// LS Electric XG5000 project: practice1
// PLC LSPLC

PROGRAM NewProgram (task: 스캔 프로그램)

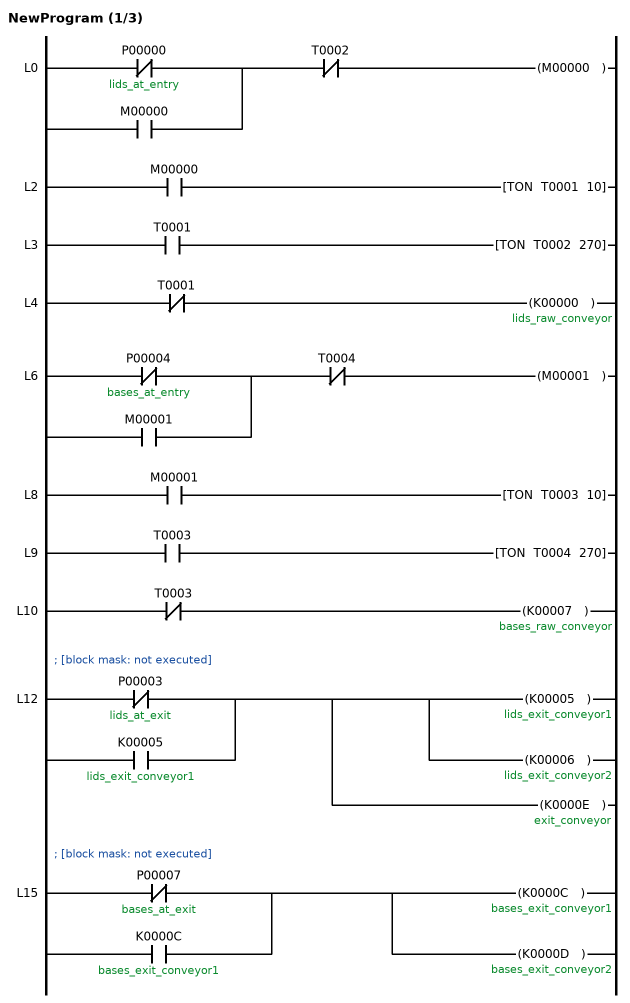
; L0
LOAD NOT  P00000	// lids_at_entry
OR        M00000
AND NOT   T0002
OUT       M00000
; L2
LOAD      M00000
TON       T0001 10
; L3
LOAD      T0001
TON       T0002 270
; L4
LOAD NOT  T0001
OUT       K00000	// lids_raw_conveyor
; L6
LOAD NOT  P00004	// bases_at_entry
OR        M00001
AND NOT   T0004
OUT       M00001
; L8
LOAD      M00001
TON       T0003 10
; L9
LOAD      T0003
TON       T0004 270
; L10
LOAD NOT  T0003
OUT       K00007	// bases_raw_conveyor
; L12 (block mask: not executed)
LOAD NOT  P00003	// lids_at_exit
OR        K00005	// lids_exit_conveyor1
OUT       K00005	// lids_exit_conveyor1
OUT       K00006	// lids_exit_conveyor2
OUT       K0000E	// exit_conveyor
; L15 (block mask: not executed)
LOAD NOT  P00007	// bases_at_exit
OR        K0000C	// bases_exit_conveyor1
OUT       K0000C	// bases_exit_conveyor1
OUT       K0000D	// bases_exit_conveyor2

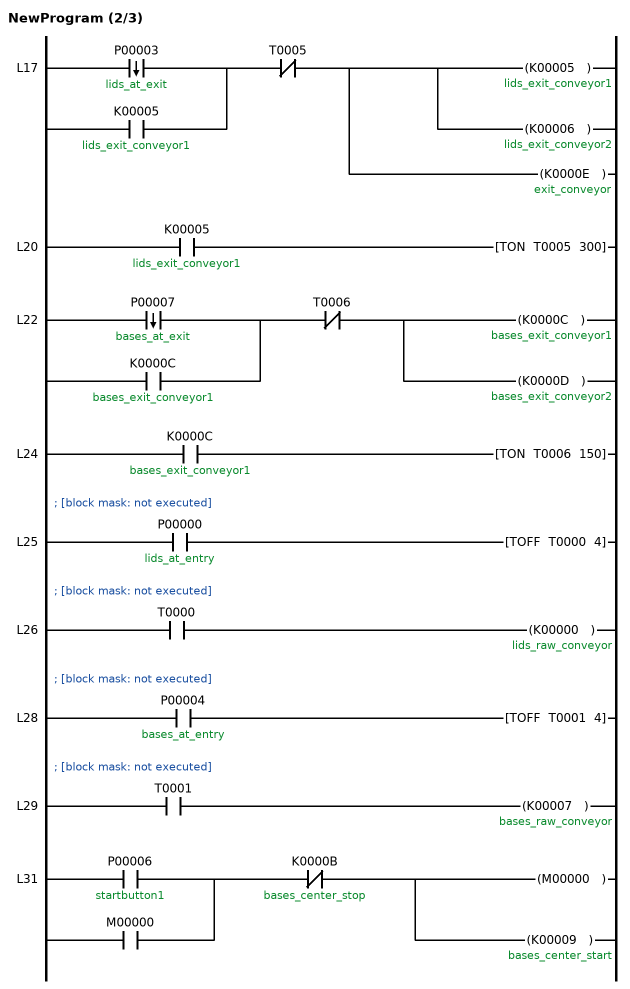
; L17
LOADN     P00003	// lids_at_exit
OR        K00005	// lids_exit_conveyor1
AND NOT   T0005
OUT       K00005	// lids_exit_conveyor1
OUT       K00006	// lids_exit_conveyor2
OUT       K0000E	// exit_conveyor
; L20
LOAD      K00005	// lids_exit_conveyor1
TON       T0005 300
; L22
LOADN     P00007	// bases_at_exit
OR        K0000C	// bases_exit_conveyor1
AND NOT   T0006
OUT       K0000C	// bases_exit_conveyor1
OUT       K0000D	// bases_exit_conveyor2
; L24
LOAD      K0000C	// bases_exit_conveyor1
TON       T0006 150
; L25 (block mask: not executed)
LOAD      P00000	// lids_at_entry
TOFF      T0000 4
; L26 (block mask: not executed)
LOAD      T0000
OUT       K00000	// lids_raw_conveyor
; L28 (block mask: not executed)
LOAD      P00004	// bases_at_entry
TOFF      T0001 4
; L29 (block mask: not executed)
LOAD      T0001
OUT       K00007	// bases_raw_conveyor
; L31
LOAD      P00006	// startbutton1
OR        M00000
AND NOT   K0000B	// bases_center_stop
OUT       M00000
OUT       K00009	// bases_center_start

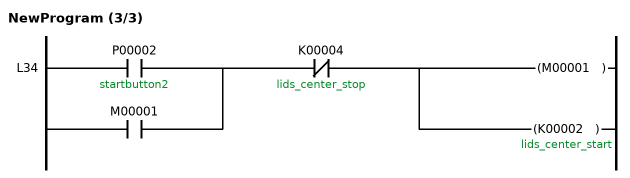
; L34
LOAD      P00002	// startbutton2
OR        M00001
AND NOT   K00004	// lids_center_stop
OUT       M00001
OUT       K00002	// lids_center_start

VARIABLES AND COMMENTS (devices not used above)
P00005	BIT	bases_center_busy
K00008	BIT	bases_center_produce_lids
K0000A	BIT	bases_center_reset
P00008	BIT	factoryio_running
P00001	BIT	lids_center_busy
K00001	BIT	lids_center_produce_lids
K00003	BIT	lids_center_reset
K0000F	BIT	lids_counter